// TIA Portal V20 export
DATA_BLOCK "Et200SpMotorstarterInterfaceHmi"   // DB208
// stored: InstanceOfName typeEt200SpMotorstarterInterfaceHmi, InstanceOfType UDT
"typeEt200SpMotorstarterInterfaceHmi"
   // VAR
   //    et200SpMotorstarterReadValue : Bool := FALSE;
   //    et200SpNumberOfMotorstarters { ExternalWritable := 'False'} : USInt := 0;
   //    et200SpUnitMotorstarter : USInt := 1;
   //    et200SpEMMotorstarter : USInt := 6;
   //    et200SpMotorstarterCurrent : Array[0.."NO_OF_ET200SPMOTORSTARTER"] of Real;
   //    et200SpMotorstarterInputs : Array[0.."NO_OF_ET200SPMOTORSTARTER"] of "LSicar_typeMotorstarterIn";
   //    et200SpMotorstarterOutputs : Array[0.."NO_OF_ET200SPMOTORSTARTER"] of "LSicar_typeMotorstarterOut";
   // END_VAR
BEGIN
   et200SpMotorstarterCurrent[0..1] := 0.0;
   et200SpMotorstarterInputs[0..1].readyAutomatic := FALSE;
   et200SpMotorstarterInputs[0..1].motorOn := FALSE;
   et200SpMotorstarterInputs[0..1].groupFault := FALSE;
   et200SpMotorstarterInputs[0..1].groupWarning := FALSE;
   et200SpMotorstarterInputs[0..1].input1 := FALSE;
   et200SpMotorstarterInputs[0..1].input2 := FALSE;
   et200SpMotorstarterInputs[0..1].input3 := FALSE;
   et200SpMotorstarterInputs[0..1].inputLocalCtrl := FALSE;
   et200SpMotorstarterInputs[0..1].iActBit0 := FALSE;
   et200SpMotorstarterInputs[0..1].iActBit1 := FALSE;
   et200SpMotorstarterInputs[0..1].iActBit2 := FALSE;
   et200SpMotorstarterInputs[0..1].iActBit3 := FALSE;
   et200SpMotorstarterInputs[0..1].iActBit4 := FALSE;
   et200SpMotorstarterInputs[0..1].iActBit5 := FALSE;
   et200SpMotorstarterInputs[0..1].manualOperating := FALSE;
   et200SpMotorstarterInputs[0..1].spare1 := FALSE;
   et200SpMotorstarterInputs[0..1].readyStartOn := FALSE;
   et200SpMotorstarterInputs[0..1].motorOnRight := FALSE;
   et200SpMotorstarterInputs[0..1].motorOnLeft := FALSE;
   et200SpMotorstarterInputs[0..1].quickstopActive := FALSE;
   et200SpMotorstarterInputs[0..1].energySaving := FALSE;
   et200SpMotorstarterInputs[0..1].moduleInserted := FALSE;
   et200SpMotorstarterInputs[0..1].exProtectionMotorActive := FALSE;
   et200SpMotorstarterInputs[0..1].blockActive := FALSE;
   et200SpMotorstarterInputs[0..1].thermalMotorOverload := FALSE;
   et200SpMotorstarterInputs[0..1].spare5 := FALSE;
   et200SpMotorstarterInputs[0..1].currentLimitTripping := FALSE;
   et200SpMotorstarterInputs[0..1].statusFailDi := FALSE;
   et200SpMotorstarterInputs[0..1].residualCurrent := FALSE;
   et200SpMotorstarterInputs[0..1].asymmetryDetected := FALSE;
   et200SpMotorstarterInputs[0..1].overtemperature := FALSE;
   et200SpMotorstarterInputs[0..1].spare7 := FALSE;
   et200SpMotorstarterOutputs[0..1].motorCw := FALSE;
   et200SpMotorstarterOutputs[0..1].motorCww := FALSE;
   et200SpMotorstarterOutputs[0..1].reserve1 := FALSE;
   et200SpMotorstarterOutputs[0..1].tripReset := FALSE;
   et200SpMotorstarterOutputs[0..1].emergencyStart := FALSE;
   et200SpMotorstarterOutputs[0..1].reserve2 := FALSE;
   et200SpMotorstarterOutputs[0..1].reserve3 := FALSE;
   et200SpMotorstarterOutputs[0..1].coldStart := FALSE;
   et200SpMotorstarterOutputs[0..1].reserve4 := FALSE;
   et200SpMotorstarterOutputs[0..1].reserve5 := FALSE;
   et200SpMotorstarterOutputs[0..1].reserve6 := FALSE;
   et200SpMotorstarterOutputs[0..1].reserve7 := FALSE;
   et200SpMotorstarterOutputs[0..1].reserve8 := FALSE;
   et200SpMotorstarterOutputs[0..1].reserve9 := FALSE;
   et200SpMotorstarterOutputs[0..1].reserve10 := FALSE;
   et200SpMotorstarterOutputs[0..1].disableQuickStop := FALSE;
END_DATA_BLOCK
